(* CoDeSys 2.3 export: NETVAROD_ACCESS_UDP.EXP *)

(* Data type *)
TYPE NetVarOD_Access_Udp :
(
	ODReadOnly,
	ODWriteOnly,
	ODReadWrite
);
END_TYPE
